// Mitsubishi GX Works2 project: group_17   PLC: FX3G

// global labels: Global1
VAR_GLOBAL
  X10_Label AT X010 : BOOL;
  X2_Label AT X002 : BOOL;
  Y5_Coil AT Y005 : BOOL;
  Oranges AT D1110 : REAL;
  Pomelos AT D1120 : REAL;
  Clememtines AT D1100 : REAL;
END_VAR
VAR_GLOBAL CONSTANT
  Multiply2 : REAL := 2;
  MultiplyHalfOranges : REAL := 0.5;
  Zero : REAL;
END_VAR
VAR_GLOBAL
  Y010_WorkDayCoil AT Y010 : BOOL;
  Orange_To_Wash AT D1130 : REAL;
END_VAR
VAR_GLOBAL CONSTANT
  hundred : REAL := 100.0;
END_VAR
VAR_GLOBAL
  Pomelos_Or_Clementines_To_Wash AT D1140 : REAL;
  TC_200 AT TC200 : BOOL;
  TS_200 AT TC200 : BOOL;
END_VAR
VAR_GLOBAL CONSTANT
  TIMER_THREE_SEC : INT := 300;
END_VAR
VAR_GLOBAL
  LEVEL2 AT M1 : BOOL;
  Coil_1 AT Y001 : BOOL;
  WashContainer AT D1180 : REAL;
  SqueezeContainer AT D1200 : REAL;
  X1_Label AT X001 : BOOL;
  M1_Label AT M1 : BOOL;
  Y001_Label AT Y001 : BOOL;
  X011_Label AT X011 : BOOL;
  X11_DoubleTap AT CC2 : BOOL;
END_VAR
VAR_GLOBAL CONSTANT
  X11_constant : WORD := 2;
END_VAR
VAR_GLOBAL
  OUT_C2 AT CS2 : BOOL;
  Y_3 AT Y003 : BOOL;
  TC_4 AT TC4 : BOOL;
END_VAR
VAR_GLOBAL CONSTANT
  TC_4_Value : WORD := 10;
END_VAR
VAR_GLOBAL
  TS_4 AT TS4 : BOOL;
  TC_5 AT TC5 : BOOL;
END_VAR
VAR_GLOBAL CONSTANT
  TC5_Val : WORD := 10;
END_VAR
VAR_GLOBAL
  TS_5 AT TS5 : BOOL;
  Y_2 AT Y002 : BOOL;
  M2_Coil AT M2 : BOOL;
  TC_2 AT TC2 : BOOL;
END_VAR
VAR_GLOBAL CONSTANT
  TC_2_Val : INT := 30;
END_VAR
VAR_GLOBAL
  TS_2 AT TS2 : BOOL;
  JuiceContainer AT D1210 : REAL;
  X3_Label AT X003 : BOOL;
  JuiceQuality AT D8281 : REAL;
END_VAR
VAR_GLOBAL CONSTANT
  GreaterThan1 : REAL := 1;
  LessThan5 : REAL := 5;
  Timer_Five_Sec : INT := 500;
END_VAR
VAR_GLOBAL
  Y4_Coil AT Y004 : BOOL;
  TC_210 AT TC210 : BOOL;
  TS_210 AT TC210 : BOOL;
  StorageContainer AT D1220 : REAL;
  CS_3 AT CS3 : BOOL;
END_VAR
VAR_GLOBAL CONSTANT
  EqualZero : REAL;
END_VAR
VAR_GLOBAL
  X_7 AT X007 : BOOL;
  M_3 AT M3 : BOOL;
  M5_Coil AT M5 : BOOL;
  CC_3 AT CC3 : BOOL;
END_VAR
VAR_GLOBAL CONSTANT
  TwoTap_X3 : WORD := 2;
END_VAR
VAR_GLOBAL
  ZeroOranges : BOOL;
  JuiceQualityVal AT D1280 : REAL;
  M_6 AT M6 : BOOL;
  M7_Coil AT M7 : BOOL;
  X_6 AT X006 : BOOL;
END_VAR
VAR_GLOBAL CONSTANT
  Min_Fiftheen : REAL := 15.0;
END_VAR
VAR_GLOBAL
  TC_250 AT TC250 : BOOL;
END_VAR
VAR_GLOBAL CONSTANT
  Timer_Ten_Sec : INT := 1000;
END_VAR
VAR_GLOBAL
  TS_250 AT TC250 : BOOL;
  TS_6 AT TS6 : BOOL;
  TC_7 AT TC7 : BOOL;
  TS_7 AT TS7 : BOOL;
  TC_8 AT TC8 : BOOL;
  TS_8 AT TS8 : BOOL;
  M8_Label AT M8 : BOOL;
  M11_Coil AT M11 : BOOL;
  M11_Label AT M11 : BOOL;
  TC_6 AT TC6 : BOOL;
  M_12 AT M12 : BOOL;
END_VAR
VAR_GLOBAL CONSTANT
  Timer_Twenty_Sec : INT := 2000;
  Div_404 : REAL := 404;
END_VAR
VAR_GLOBAL
  JuiceQualityInput AT D8281 : INT;
END_VAR
VAR_GLOBAL CONSTANT
  EqualZeroInt : INT;
END_VAR
VAR_GLOBAL
  Y_0 AT Y000 : BOOL;
  M_13 AT M13 : BOOL;
  X_5 AT X005 : BOOL;
END_VAR
VAR_GLOBAL CONSTANT
  Mul_73 : REAL := 73;
END_VAR
VAR_GLOBAL
  MinimumValue AT D8282 : INT;
  Pomelos_To_Wash AT D1140 : REAL;
  Clementines_To_Wash AT D1290 : REAL;
END_VAR

// task Task_01 (event TRUE, interval 0, priority 31): POU_01

PROGRAM POU_01
(* structured ladder/FBD written out as ST: instructions are called as NAME(EN, inputs, outputs); _pN, _eN, _tN stand for wires *)
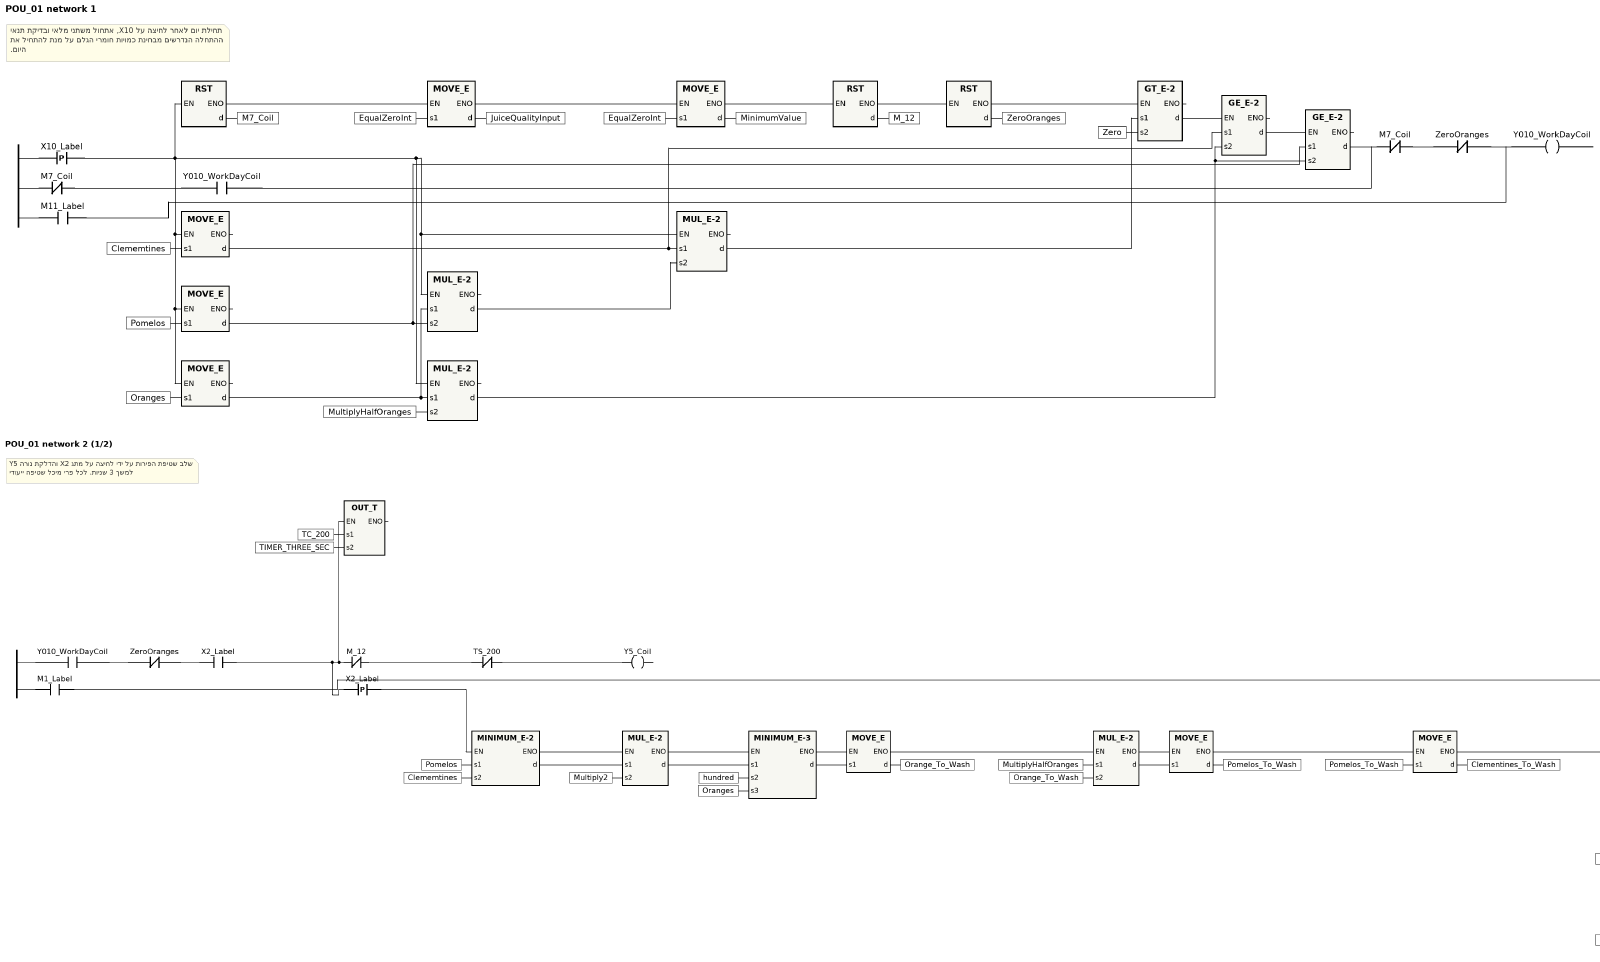
(* network 1 *)
(* תחילת יום לאחר לחיצה על X10, אתחול משתני מלאי ובדיקת תנאי ההתחלה הנדרשים מבחינת כמויות חומרי הגלם על מנת להתחיל את היום. *)
_p1 := LDP(TRUE, X10_Label);
_e2 := RST(_p1, M7_Coil);
_e3 := MOVE_E(_e2, EqualZeroInt, JuiceQualityInput);
_e4 := MOVE_E(_e3, EqualZeroInt, MinimumValue);
_e5 := RST(_e4, M_12);
_e6 := RST(_e5, ZeroOranges);
MOVE_E(_p1, Oranges, _t7);
MUL_E(_p1, _t7, MultiplyHalfOranges, _t8);
MOVE_E(_p1, Clememtines, _t9);
MOVE_E(_p1, Pomelos, _t10);
MUL_E(_p1, _t7, _t10, _t11);
MUL_E(_p1, _t9, _t11, _t12);
GT_E(_e6, _t12, Zero, _t13);
GE_E(_t13, _t9, _t8, _t14);
GE_E(_t14, _t10, _t8, _t15);
Y010_WorkDayCoil := (((_t15 OR (NOT M7_Coil AND Y010_WorkDayCoil)) AND NOT M7_Coil) AND NOT ZeroOranges) OR M11_Label;
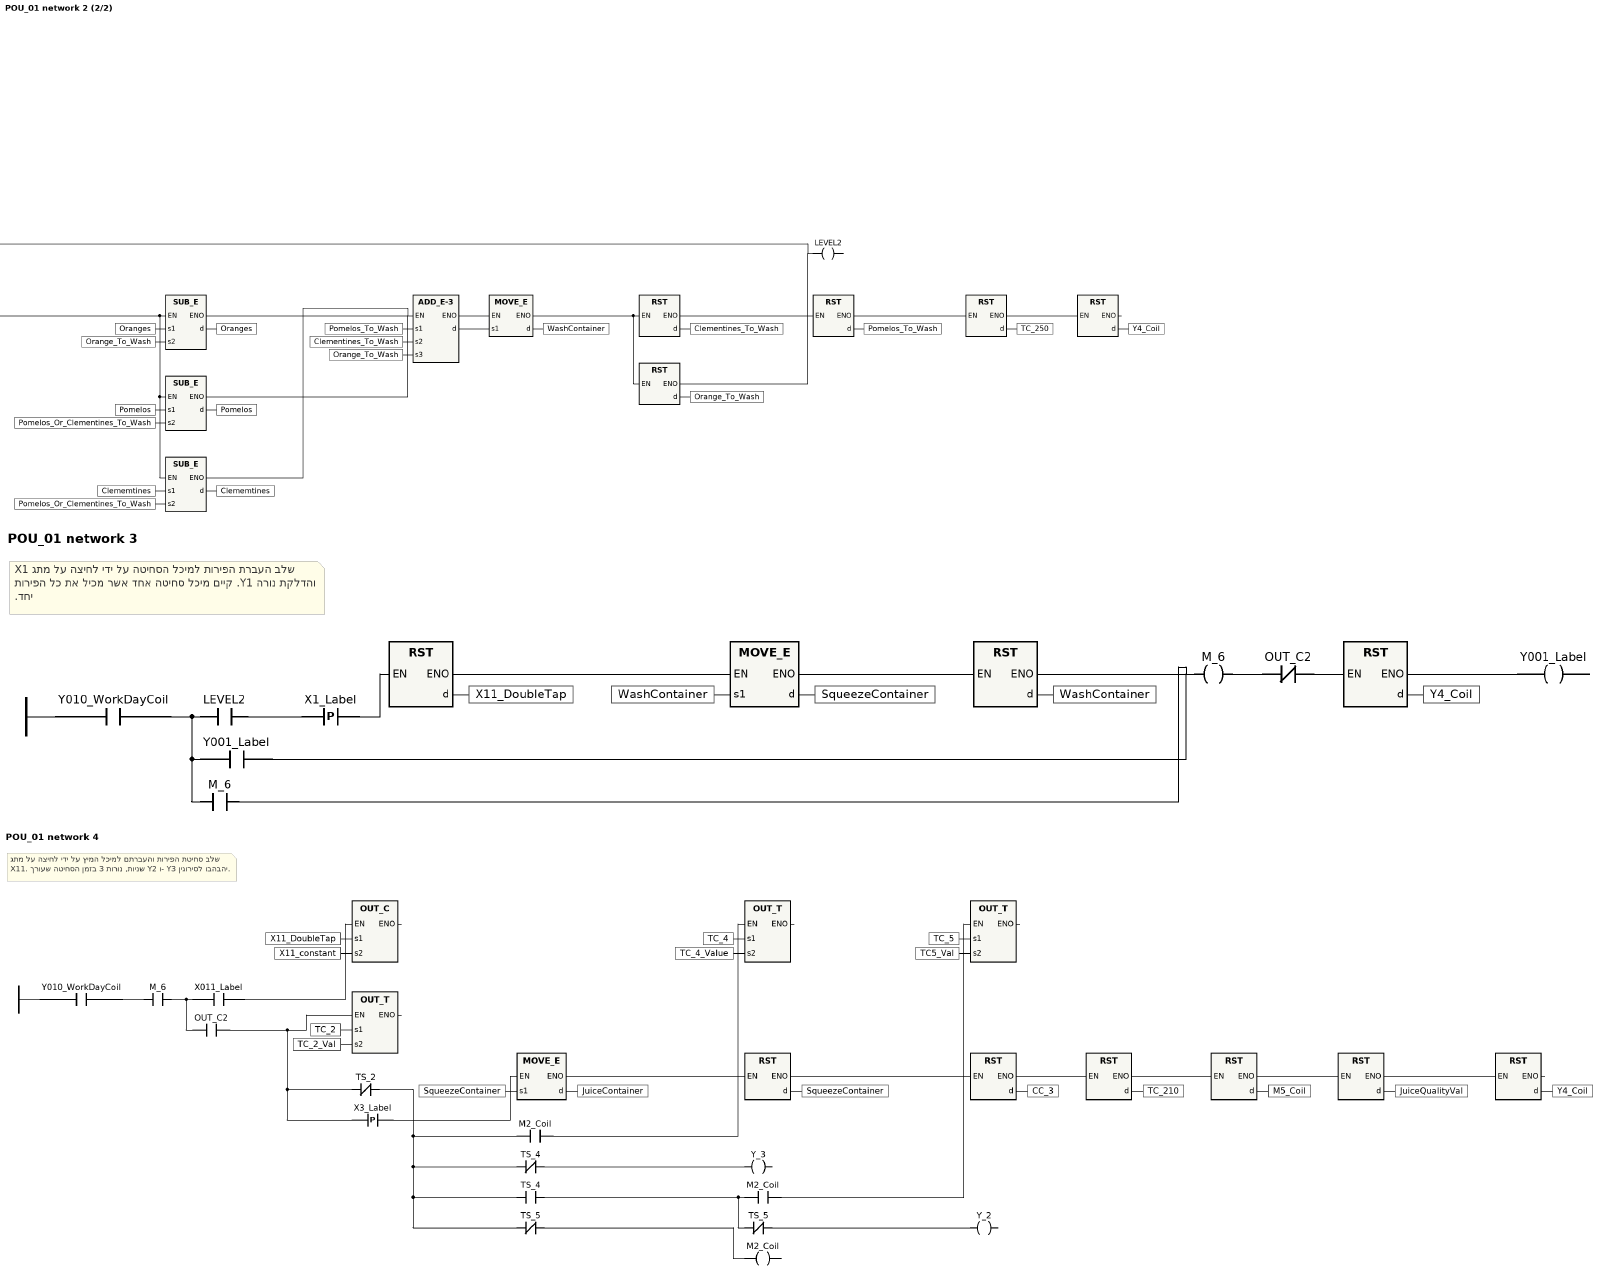
(* network 2 *)
(* שלב שטיפת הפירות על ידי לחיצה על מתג X2 והדלקת נורה Y5 למשך 3 שניות. לכל פרי מיכל שטיפה ייעודי *)
_p1 := Y010_WorkDayCoil AND NOT ZeroOranges AND X2_Label;
OUT_T(_p1, TC_200, TIMER_THREE_SEC);
Y5_Coil := _p1 AND NOT M_12 AND NOT TS_200;
_e3 := MINIMUM_E(_p1 AND LDP(TRUE, X2_Label), Pomelos, Clememtines, _t2);
_e5 := MUL_E(_e3, _t2, Multiply2, _t4);
_e7 := MINIMUM_E(_e5, _t4, hundred, Oranges, _t6);
_e8 := MOVE_E(_e7, _t6, Orange_To_Wash);
_e10 := MUL_E(_e8, MultiplyHalfOranges, Orange_To_Wash, _t9);
_e11 := MOVE_E(_e10, _t9, Pomelos_To_Wash);
_e12 := MOVE_E(_e11, Pomelos_To_Wash, Clementines_To_Wash);
_e13 := SUB_E(_e12, Oranges, Orange_To_Wash, Oranges);
_e14 := SUB_E(_e12, Pomelos, Pomelos_Or_Clementines_To_Wash, Pomelos);
_e15 := SUB_E(_e12, Clememtines, Pomelos_Or_Clementines_To_Wash, Clememtines);
_e17 := ADD_E(_e13 OR _e14 OR _e15, Pomelos_To_Wash, Clementines_To_Wash, Orange_To_Wash, _t16);
_e18 := MOVE_E(_e17, _t16, WashContainer);
_e19 := RST(_e18, Clementines_To_Wash);
_e20 := RST(_e19, Pomelos_To_Wash);
_e21 := RST(_e20, TC_250);
RST(_e21, Y4_Coil);
_e22 := RST(_e18, Orange_To_Wash);
LEVEL2 := _e22 OR M1_Label;
(* network 3 *)
(* שלב העברת הפירות למיכל הסחיטה על ידי לחיצה על מתג X1 והדלקת נורה Y1. קיים מיכל סחיטה אחד אשר מכיל את כל הפירות יחד. *)
_e1 := RST(Y010_WorkDayCoil AND LEVEL2 AND LDP(TRUE, X1_Label), X11_DoubleTap);
_e2 := MOVE_E(_e1, WashContainer, SqueezeContainer);
_e3 := RST(_e2, WashContainer);
_p4 := _e3 OR (Y010_WorkDayCoil AND Y001_Label) OR (Y010_WorkDayCoil AND M_6);
M_6 := _p4;
_e5 := RST(_p4 AND NOT OUT_C2, Y4_Coil);
Y001_Label := _e5;
(* network 4 *)
(* שלב סחיטת הפירות והעברתם למיכל המיץ על ידי לחיצה על מתג X11. בזמן הסחיטה שעורך 3 שניות, נורות Y2 ו- Y3 יהבהבו לסירוגין. *)
_p1 := Y010_WorkDayCoil AND M_6;
OUT_C(_p1 AND X011_Label, X11_DoubleTap, X11_constant);
_p2 := _p1 AND OUT_C2;
OUT_T(_p2, TC_2, TC_2_Val);
_p3 := _p2 AND NOT TS_2;
OUT_T(_p3 AND M2_Coil, TC_4, TC_4_Value);
Y_3 := _p3 AND NOT TS_4;
_p4 := _p3 AND TS_4;
OUT_T(_p4 AND M2_Coil, TC_5, TC5_Val);
Y_2 := _p4 AND NOT TS_5;
M2_Coil := _p3 AND NOT TS_5;
_e5 := MOVE_E(_p2 AND LDP(TRUE, X3_Label), SqueezeContainer, JuiceContainer);
_e6 := RST(_e5, SqueezeContainer);
_e7 := RST(_e6, CC_3);
_e8 := RST(_e7, TC_210);
_e9 := RST(_e8, M5_Coil);
_e10 := RST(_e9, JuiceQualityVal);
RST(_e10, Y4_Coil);
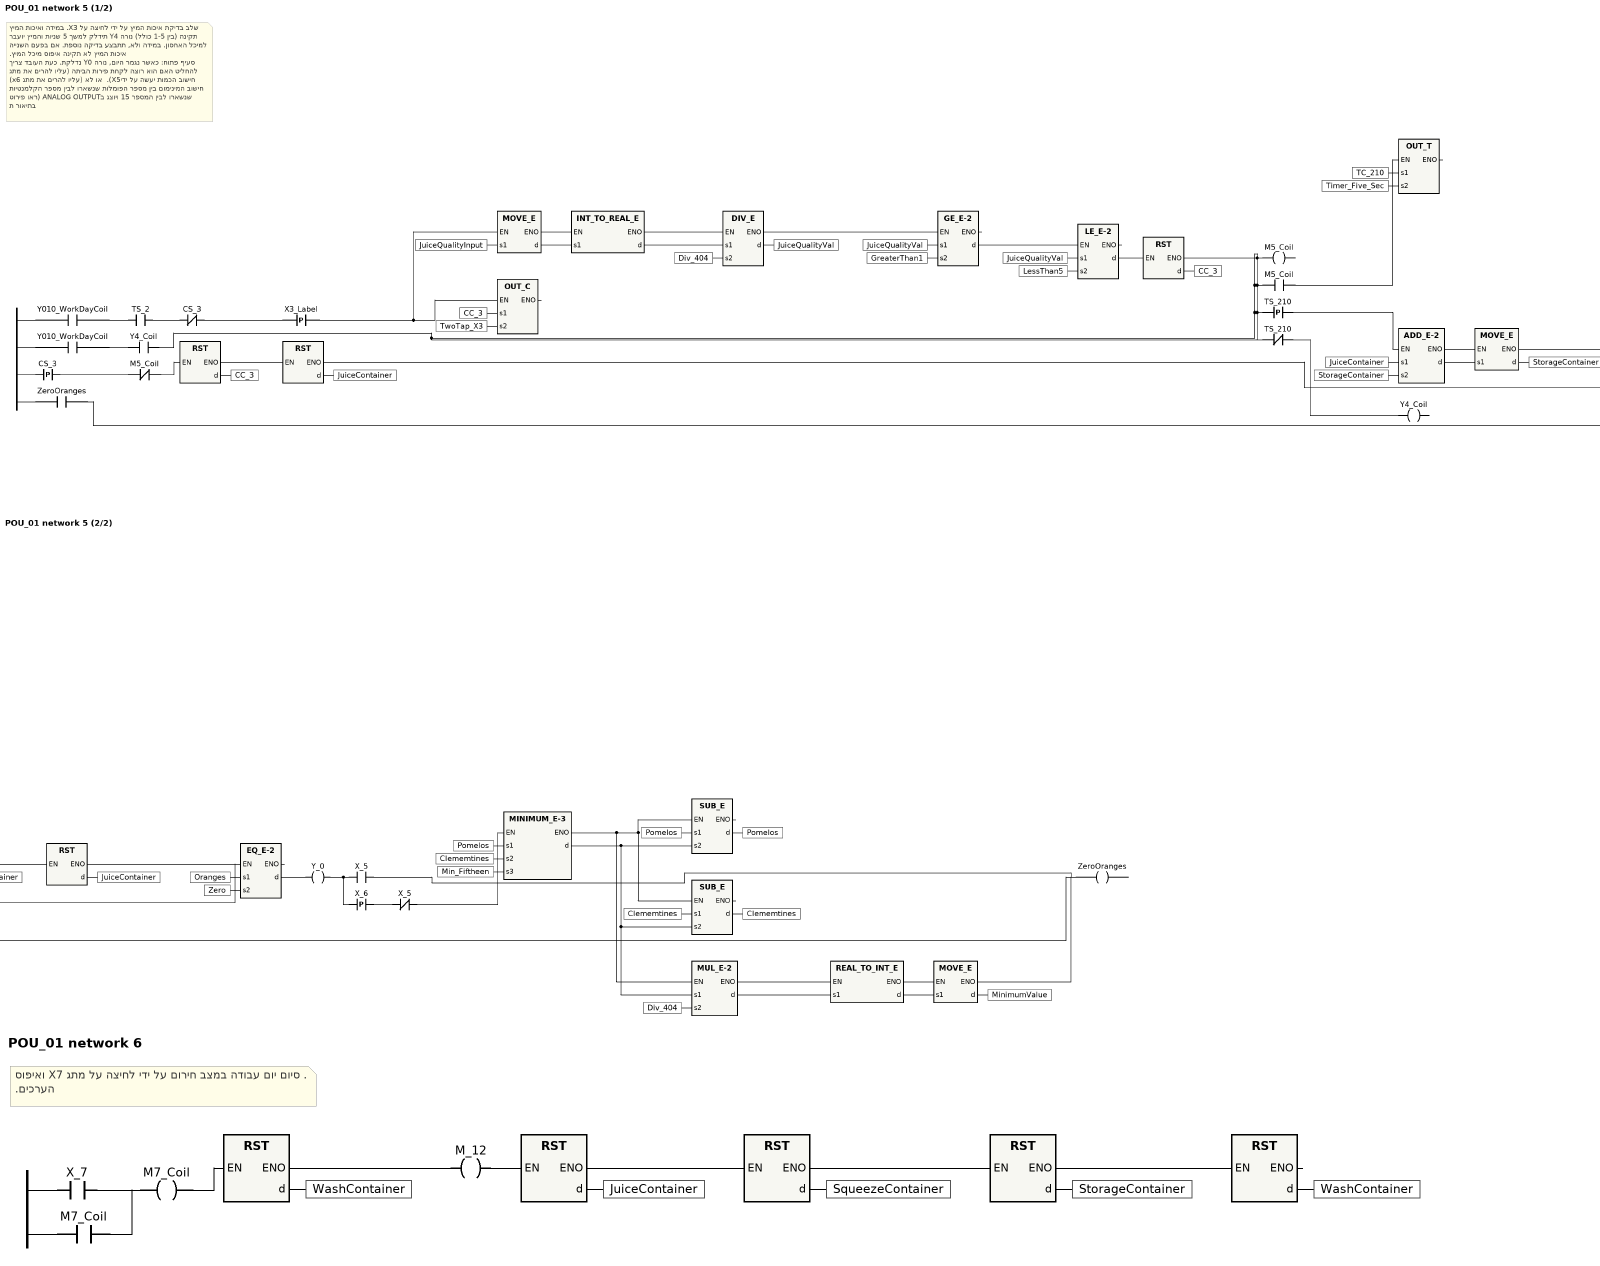
(* network 5 *)
(* שלב בדיקת איכות המיץ על ידי לחיצה על X3. במידה ואיכות המיץ תקינה (בין 1-5 כולל) נורה Y4 תידלק למשך 5 שניות והמיץ יועבר למיכל האחסון. במידה ולא, תתבצע בדיקה נוספת. אם בפעם השנייה איכות המיץ לא תקינה איפוס מיכל המיץ.  / סעיף פתוח: כאשר נגמר היום, נורה Y0 נדלקת. כעת העובד צריך להחליט האם הוא רוצה לקחת פירות הביתה (עליו להרים את מתג (x6 או לא (עליו להרים את מתג  .(X5חישוב הכמות יעשה על ידי חישוב המינימום בין מספר הפומלות שנשארו לבין מספר הקלמנטיות שנשארו לבין המספר 15 ויוצג בANALOG OUTPUT (ראו פירוט בתיאור ת *)
_p1 := Y010_WorkDayCoil AND TS_2 AND NOT CS_3 AND LDP(TRUE, X3_Label);
_e3 := MOVE_E(_p1, JuiceQualityInput, _t2);
_e5 := INT_TO_REAL_E(_e3, _t2, _t4);
_e6 := DIV_E(_e5, _t4, Div_404, JuiceQualityVal);
GE_E(_e6, JuiceQualityVal, GreaterThan1, _t7);
LE_E(_t7, JuiceQualityVal, LessThan5, _t8);
_e9 := RST(_t8, CC_3);
_p10 := _e9 OR (Y010_WorkDayCoil AND Y4_Coil);
M5_Coil := _p10;
OUT_C(_p1, CC_3, TwoTap_X3);
OUT_T(_p10 AND M5_Coil, TC_210, Timer_Five_Sec);
_e12 := ADD_E(_p10 AND LDP(TRUE, TS_210), JuiceContainer, StorageContainer, _t11);
_e13 := MOVE_E(_e12, _t11, StorageContainer);
_e14 := RST(_e13, JuiceContainer);
Y4_Coil := _p10 AND NOT TS_210;
_e15 := RST(LDP(TRUE, CS_3) AND NOT M5_Coil, CC_3);
_e16 := RST(_e15, JuiceContainer);
EQ_E(_e14 OR _e16, Oranges, Zero, _t17);
Y_0 := _t17;
_e19 := MINIMUM_E(_t17 AND LDP(TRUE, X_6) AND NOT X_5, Pomelos, Clememtines, Min_Fiftheen, _t18);
_e21 := MUL_E(_e19, _t18, Div_404, _t20);
_e23 := REAL_TO_INT_E(_e21, _t20, _t22);
_e24 := MOVE_E(_e23, _t22, MinimumValue);
ZeroOranges := (_t17 AND X_5) OR _e24 OR ZeroOranges;
SUB_E(_e19, Pomelos, _t18, Pomelos);
SUB_E(_e19, Clememtines, _t18, Clememtines);
(* network 6 *)
(* . סיום יום עבודה במצב חירום על ידי לחיצה על מתג X7 ואיפוס הערכים. *)
_p1 := X_7 OR M7_Coil;
M7_Coil := _p1;
_e2 := RST(_p1, WashContainer);
M_12 := _e2;
_e3 := RST(_e2, JuiceContainer);
_e4 := RST(_e3, SqueezeContainer);
_e5 := RST(_e4, StorageContainer);
RST(_e5, WashContainer);
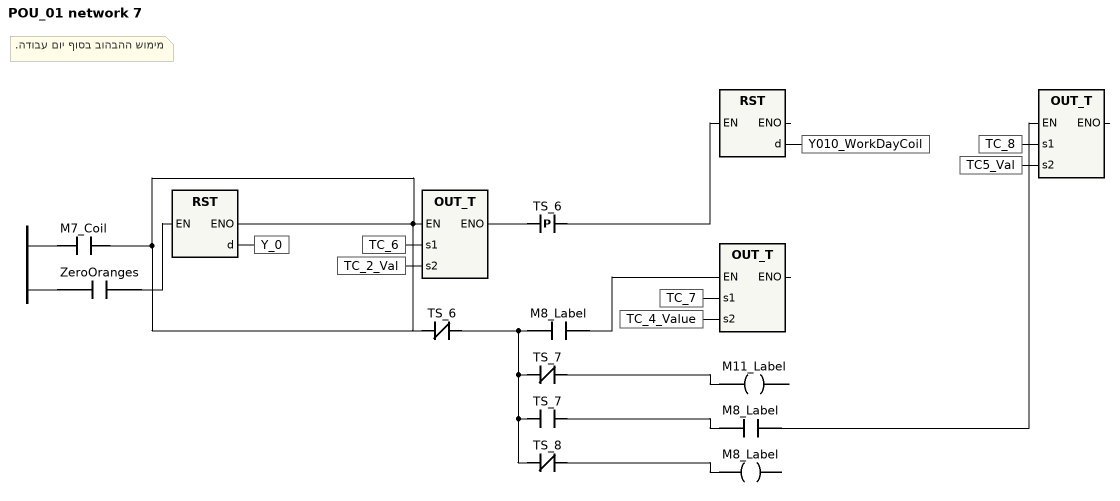
(* network 7 *)
(* מימוש ההבהוב בסוף יום עבודה. *)
_e1 := RST(ZeroOranges, Y_0);
_p2 := M7_Coil OR _e1;
_e3 := OUT_T(_p2, TC_6, TC_2_Val);
RST(_e3 AND LDP(TRUE, TS_6), Y010_WorkDayCoil);
_p4 := _p2 AND NOT TS_6;
OUT_T(_p4 AND M8_Label, TC_7, TC_4_Value);
M11_Label := _p4 AND NOT TS_7;
OUT_T(_p4 AND TS_7 AND M8_Label, TC_8, TC5_Val);
M8_Label := _p4 AND NOT TS_8;
END_PROGRAM
